PROGRAM MAIN
VAR
	fbCylinderTest : FB_CylinderTest;
	fbTest : FB_FuseTest;
	fbTest1 : FB_EL922x_ChannelExtended;
	fbTest2 : FB_EL922x_ChannelExtended;
	xTes: BOOL;
	xTest1: BOOL;
	switched: BOOL;
	xTest2: BOOL;
END_VAR

//tcUnit.RUN();
fbTest();

IF xTes THEN
	fbTest.METH(chn1 := fbTest1, chn2 := fbTest2);
	xTes := false;
END_IF
IF xTest1 THEN
	switched := fbTest.GetDisabledBySwitch();
	xTest1 := FALSE;
END_IF

IF xTest2 THEN
	fbTest.SwitchChannel1();
	xTest2 := FALSE;
END_IF

END_PROGRAM

(* stored: Version 1.1.0.1, ProductVersion 3.1.4024.5
   POU MAIN: Id {f20f72a3-44bd-4b01-bab9-6aeb1376a30d}, SpecialFunc None *)
